// TIA Portal V17 export
// export: Created 2024-06-27T19:41:44.5933912Z, ExportSetting WithDefaults, DisplayName Totally Integrated Automation Portal, DisplayVersion V17, DisplayName TIA Portal Openness, DisplayVersion V17, DisplayName TIA Portal Version Control Interface, DisplayVersion V17, DisplayName STEP 7 Professional, DisplayVersion V17, DisplayName STEP 7 Safety, DisplayVersion V17, DisplayName WinCC Professional, DisplayVersion V17
DATA_BLOCK "RCT"   // DB1005
{ S7_Optimized_Access := 'TRUE' }
VERSION : 0.1
// stored: AutoNumber false, DBAccessibleFromOPCUA true, DBAccessibleFromWebserver true, IsOnlyStoredInLoadMemory false, IsRetainMemResEnabled false, IsWriteProtectedInAS false, MemoryReserve 100
   VAR
      St2 : Struct
         Axe_X1 : Struct
            Vel_Vision : LReal;
            Pos_Vision : LReal;
            ModeAbs : Bool;
            ModeRel : Bool;
         END_STRUCT;
         Prehenseur_Z : Struct
            Pos_Vision : LReal;
         END_STRUCT;
         Autorisation_Vision : Bool;
         Fin_Vision : Bool;
      END_STRUCT;
      St3 : Struct
         Axe_X1 : Struct
            Vel_RX : LReal;
            Pos_RX : LReal;
            ModeAbs : Bool;
            ModeRel : Bool;
         END_STRUCT;
         Axe_Y : Struct
            Pos_RX : LReal;
         END_STRUCT;
         Axe_Z : Struct
            Pos_RX : LReal;
         END_STRUCT;
         Autorisation_RX : Bool;
         Fin_RX : Bool;
      END_STRUCT;
      St4 : Struct
         Axe_X1 : Struct
            Pos_Marquage : LReal;
         END_STRUCT;
         Axe_Y1 : Struct
            Pos_Marquage : LReal;
         END_STRUCT;
      END_STRUCT;
   END_VAR
BEGIN
END_DATA_BLOCK
